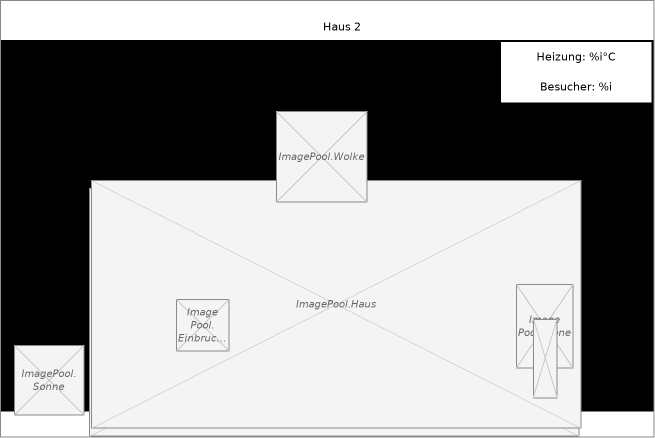
VISUALIZATION Haus_2  // 655x438
    Rectangle (1,40 652x371)
    Rectangle (1,40 652x371), colour variable: L_Himmel
        p2167032090: L_Himmel
    Image (89,188 490x248), image: ImagePool.Licht
        p84334746: Haus2.BildLicht
    Image (91,180 490x248), image: ImagePool.Haus
    Image (516,284 57x84), image: ImagePool.Krone
        p2858320360: L_Baum
    Image (533,319 24x79), image: ImagePool.Stamm
    Image (14,345 70x70), image: ImagePool.Sonne
        p2858320360: L_Sonnenstand
        p84334746: L_Sonne
    Image (176,299 53x52), image: ImagePool.Einbruch_grun
        p84334746: Haus2.L_EinbruchBild
    Image (276,111 91x91), image: ImagePool.Wolke
        p84334746: Haus2.WetterBild
    Textfield (267,16 150x22), "Haus 2"
    Textfield (501,42 150x30), "Heizung: %i°C", text variable: net_heizung_02
    Textfield (501,72 150x30), "Besucher: %i", text variable: net_besucher_02
END_VISUALIZATION

(* stored: Version 1.1.0.1, ProductVersion 3.1.4018.5
   Visu Haus_2: Id {417285eb-4cc9-41fe-bb70-cd8f0d66752b} *)
